TYPE ST_TorchAdsStruct :
STRUCT
	bMainSwitch			: BOOL;
	bAutoSwitch	   		: BOOL;
	bStartButton   		: BOOL;
	bStopButton	   		: BOOL;
	bResetButton   		: BOOL;
	rPosition	   		: REAL;
	rPreassure	   		: REAL;
	wWorkTimeHours  	: UDINT;
	wWorkTimeMinutes    : UINT;	
	wWorkTimeSeconds    : UINT;
	wStatus		   		: WORD;
	iIgnitCount			: UDINT;
	sStateLabel    		: T_MaxString;
	sStatusLabel   		: T_MaxString;
	
END_STRUCT
END_TYPE

(* stored: Version 1.1.0.1, ProductVersion 3.1.4024.15
   DUT ST_TorchAdsStruct: Id {6eb22e63-53a0-4c10-9d57-86541dfb99b5} *)
